// TIA Portal V17 export
// export: Created 2024-10-17T14:16:17.7123061Z, ExportSetting WithDefaults, DisplayName Totally Integrated Automation Portal, DisplayVersion V17 Update 4, DisplayName TIA Portal Openness, DisplayVersion V17 Update 4, DisplayName TIA Portal Version Control Interface, DisplayVersion V17, DisplayName SINAMICS Startdrive Advanced, DisplayVersion V17 Update2, DisplayName SINAMICS Startdrive G130, G150, S120, S150, SINAMICS MV, S210, DisplayVersion V17 Update2, DisplayName SINAMICS Startdrive G110M, G120, G120C, G120D, G120P, G115D, DisplayVersion V17 Update2, DisplayName STEP 7 Professional, DisplayVersion V17 Update 4, DisplayName STEP 7 Safety, DisplayVersion V17, DisplayName WinCC Advanced / Unified PC, DisplayVersion V17 Update 4
TYPE "LPMLV2022_typeEvent"
TITLE = LPMLV2022_typeEvent
// Support: tech.team.motioncontrol@siemens.com
// stored: IsFailsafeCompliant false
   STRUCT
      Trigger { ExternalWritable := 'False'} : Bool;   // Alarm Message Trigger. Alarm trigger should be turned on only when the alarm is currently active
      ID { ExternalWritable := 'False'} : DInt;   // Alarm Message Identification Number. The alarm ID number is a unique value assigned to each alarm. Minimum required for information/machine monitoring
      Value { ExternalWritable := 'False'} : DInt;   // Alarm Message Number. The alarm message number is a value that is associated to the alarm allowing for user specific detail or to break down the Alarm.ID to greater detail
      Message { ExternalWritable := 'False'} : String[80];   // Alarm Message. The alarm message is the actual text of the alarm for those machines capable of providing string information
      Category { ExternalWritable := 'False'} : DInt;   // Alarm Category. Alarm category is used to identity what type of alarm has occurred (e.g. electrical, mechanical, materials, utilities, etc.)
      DateTime { ExternalWritable := 'False'} : "LPMLV2022_typeDateTime";   // Date and Time the Alarm Occurred. The timestamp for when the alarm was first triggered
      DateTimeDTL { ExternalWritable := 'False'} : DTL;   // Date and Time (DTL) the Alarm Occurred. The timestamp for when the alarm was first triggered
      AckDateTime { ExternalWritable := 'False'} : "LPMLV2022_typeDateTime";   // Date and Time the Alarm was Acknowledged. The timestamp for when the alarm was acknowledged by the operator, or cleared
      AckDateTimeDTL { ExternalWritable := 'False'} : DTL;   // Date and Time (DTL) the Alarm was Acknowledged. The timestamp for when the alarm was acknowledged by the operator, or cleared
   END_STRUCT;
END_TYPE
